TEXTLIST ButtonStates
  0 = 'Enable'
  1 = 'Disable'
   = ''
END_TEXTLIST

(* stored: Version 1.1.0.1, ProductVersion 3.1.4022.12
   TextList ButtonStates: Id {537763f7-a462-4fc7-b16e-19856dde75d8} *)
